{attribute 'qualified_only'}
VAR_GLOBAL
	motorR: AXIS_REF;
	motorL: AXIS_REF;
	coderR: AXIS_REF;
	coderL: AXIS_REF;
	
	lrPosX: LREAL;
	lrPosY: LREAL;
	lrAngle: LREAL;
	
	
END_VAR

(* stored: Version 1.1.0.1, ProductVersion 3.1.4022.18
   GVL Motors: Id {5510c189-5108-43cc-8296-1cc82dc26db4} *)
